FUNCTION rotZ : mat3d
VAR_IN_OUT CONSTANT
	i_mat : Mat3d;
	i_ang : LREAL;
END_VAR
VAR
	rot :Mat3d := g_eye3d;
END_VAR

rot[1,1]:=COS(i_ang);
rot[2,2]:=rot[1,1];
rot[2,1]:=SIN(i_ang);
rot[1,2]:=-rot[2,1];
matMultiply(i_mat, rot, rotZ);

END_FUNCTION

(* stored: Version 1.1.0.1, ProductVersion 3.1.4024.12
   POU rotZ: Id {1bf0182b-424b-4cd5-a62f-6a71e23fd9fa}, SpecialFunc None *)
